Fanuc KAREL source: kt00002.KL

-- PROVISIONAL review KL for V940-1; original PC SHA256 d48bb7cb35c718279e7b6bea9bafd8ccc0777e7f6a9ef6330707a90f35a8935b
-- Incomplete behavior may be omitted. Consult companion uncertainty JSON. Do not deploy.
PROGRAM KT00002
%NOLOCKGROUP
VAR
  I1 : INTEGER
  I2 : INTEGER
  OUT : REAL
BEGIN
  -- V9_ZERO_TABLE_METADATA_HINT layout=0001; no indexed target words; source/name/runtime held
  -- UNRESOLVED_PC offsets 5-16; opcodes 2E,23
  -- UNRESOLVED_PC offsets 21-32; opcodes 2E,23
  -- UNRESOLVED_PC offsets 37-48; opcodes 2E,23
  -- UNRESOLVED_PC offsets 53-64; opcodes 2E,23
  -- UNRESOLVED_PC offsets 69-89; opcodes 21,21,52,64,23
  -- UNRESOLVED_PC offsets 94-98; opcodes 7F
END KT00002
